PROGRAM MAIN
VAR
	myCsvWriter : CSVWriter;
	myJsonWriter : JsonWriter;
	myTextWriter : TextWriter;
	myObject : SomeCyclicClass := (MyWriter := myTextWriter);
	runOperation1: BOOL;
	runOperation2: BOOL;
	runOperation3: BOOL;
	xtest: BOOL;
END_VAR

IF runOperation1 THEN
	runOperation1 := FALSE;
	myObject.MyWriter := myJsonWriter;
	myObject.DoSomething();
END_IF

IF runOperation2 THEN
	runOperation2 := FALSE;
	myObject.MyWriter := myTextWriter;
	myObject.DoSomething();
END_IF

IF runOperation3 THEN
	runOperation3 := FALSE;
	myObject.MyWriter := myCsvWriter;
	myObject.DoSomething();
END_IF

IF xtest THEN
	xtest := FALSE;
	myObject.MyWriter := myCsvWriter;
END_IF

END_PROGRAM

(* stored: Version 1.1.0.1, ProductVersion 3.1.4024.12
   POU MAIN: Id {46c6e83c-31ed-463f-8e37-5ce86575fcba}, SpecialFunc None *)
